// TIA Portal V16 export
// export: Created 2020-10-15T12:04:38.5046435Z, ExportSetting WithDefaults, DisplayName Totally Integrated Automation Portal, DisplayVersion V16, DisplayName TIA Portal Version Control Interface, DisplayVersion V16, DisplayName TIA Portal Openness, DisplayVersion V16, DisplayName STEP 7 Professional, DisplayVersion V16, DisplayName STEP 7 Safety, DisplayVersion V16, DisplayName WinCC Advanced, DisplayVersion V16
VAR_GLOBAL   // PLC tag table "Euchner"
   "001WAS001_PI_F" AT %I80.0 : "iUDT_PI_F_WAS";   // Periphery interface failsafe inputs VI cleaning switch / Peripherieschnittstelle sichere Eingänge -VI Reinigungsschalter
   "001WAS001_PI" AT %I88.0 : "iUDT_PI_WAS";   // Periphery interface inputs VI cleaning switch / Peripherieschnittstelle Eingänge -VI Reinigungschalter
   "001WAS001_PO" AT %Q88.0 : "iUDT_PO_WAS";   // Periphery interface outputs VI cleaning switch / Peripherieschnittstelle Ausgänge -VI Reinigungschalter
   "010STU001_PI_F" AT %I2510.0 : "iUDT_PI_F_STU";   // Periphery interface failsafe inputs Euchner box / Schutztür sichere Peripherieeingänge
   "010STU001_PO_F" AT %Q2510.0 : "iUDT_PO_F_STU";   // Safety door safety periphery outputs / Schutztür sichere Peripherieausgänge
   "010STU001_PI" AT %I2500.0 : "iUDT_PI_STU";   // Periphery interface inputs Euchner box / Schutztür Peripherieeingänge
   "010STU001_PO" AT %Q2500.0 : "iUDT_PO_STU";   // Safety door periphery outputs / Schutztür Peripherieausgänge
   "020STU001_PI_F" AT %I2530.0 : "iUDT_PI_F_STU";   // Periphery interface failsafe inputs Euchner box / Schutztür sichere Peripherieeingänge
   "020STU001_PO_F" AT %Q2530.0 : "iUDT_PO_F_STU";   // Safety door safety periphery outputs / Schutztür sichere Peripherieausgänge
   "020STU001_PI" AT %I2520.0 : "iUDT_PI_STU";   // Periphery interface inputs Euchner box / Schutztür Peripherieeingänge
   "020STU001_PO" AT %Q2520.0 : "iUDT_PO_STU";   // Safety door periphery outputs / Schutztür Peripherieausgänge
   "020STU002_PI_F" AT %I2550.0 : "iUDT_PI_F_STU";   // Periphery interface failsafe inputs Euchner box / Schutztür sichere Peripherieeingänge
   "020STU002_PO_F" AT %Q2550.0 : "iUDT_PO_F_STU";   // Safety door safety periphery outputs / Schutztür sichere Peripherieausgänge
   "020STU002_PI" AT %I2540.0 : "iUDT_PI_STU";   // Periphery interface inputs Euchner box / Schutztür Peripherieeingänge
   "020STU002_PO" AT %Q2540.0 : "iUDT_PO_STU";   // Safety door periphery outputs / Schutztür Peripherieausgänge
   "050STU001_PI_F" AT %I2570.0 : "iUDT_PI_F_STU";   // Periphery interface failsafe inputs Euchner box / Schutztür sichere Peripherieeingänge
   "050STU001_PO_F" AT %Q2570.0 : "iUDT_PO_F_STU";   // Safety door safety periphery outputs / Schutztür sichere Peripherieausgänge
   "050STU001_PI" AT %I2560.0 : "iUDT_PI_STU";   // Periphery interface inputs Euchner box / Schutztür Peripherieeingänge
   "050STU001_PO" AT %Q2560.0 : "iUDT_PO_STU";   // Safety door periphery outputs / Schutztür Peripherieausgänge
   "010STU001-Errorword" AT %IW2504 : Word;   // Schutztür Fehlerword
   "020STU001-Errorword" AT %IW2524 : Word;   // Schutztür Fehlerword
   "020STU002-Errorword" AT %IW2544 : Word;   // Schutztür Fehlerword
   "050STU001-Errorword" AT %IW2564 : Word;   // Schutztür Fehlerword
END_VAR
